(* IEC 61131-3 sources: LASAL/Class/SendNow, 1 file *)

(* ---- SendNow.st ---- *)
(*!
<Class
	Name               = "SendNow"
	Revision           = "0.0"
	RealtimeTask       = "false"
	CyclicTask         = "false"
	BackgroundTask     = "false"
	Sigmatek           = "false"
	OSInterface        = "false"
	HighPriority       = "false"
	Automatic          = "false"
	UpdateMode         = "Prescan"
	SharedCommandTable = "true"
	Objectsize         = "(390,120)">
	<Channels>
		<Server Name="ClassSvr" Visualized="false" Initialize="false" WriteProtected="true" Retentive="false"/>
		<Client Name="CommandServer" Required="true" Internal="false"/>
	</Channels>
</Class>
*)
SendNow : CLASS
  //Servers:
	ClassSvr 	: SvrChCmd_DINT;
  //Clients:
	CommandServer 	: CltChCmd_CommandServer;
  //Variables:
  //Functions:
  //Tables:
	FUNCTION @STD
		VAR_OUTPUT
			ret_code	: CONFSTATES;
		END_VAR;
	FUNCTION GLOBAL TAB @CT_;
END_CLASS;

#pragma usingLtd CommandServer
